Universal Robots PolyScope program: 8_put_glass_down.urp

Program 8_put_glass_down (installation=default directory=/programs/washer_rahman createdIn=5.9.5.1031259 lastSavedIn=5.9.5.1031259 robotSerialNumber=20215500597)
Calibrated DH parameters: a=[0.000193, -0.066673, -0.391568, -0.000012, 0.00005, 0]; d=[0.162643, -472.05677, 465.132521, 7.058239, 0.099746, 0.099582]; alpha=[1.571116, 0.00089, 0.003862, 1.569269, -1.569248, 0]; deltaTheta=[0, -1.413394, 7.628392, 0.068187, 0, -0.000001]
Robot Program (runOnlyOnce=true)
  SuppressedNode
    var_2 := 3
  SuppressedNode
    Script: glass_hover=p[-.603,-0.23+var_2*0.150 ,0.277,2.067,2.652,-2.043]
  Script: glass_hover=p[-.603,-0.23+GP_int_in[0]*0.150 ,0.277,2.067,2.652,-2.043]
  MoveJ speed 60 deg/s, acceleration 80 deg/s^2 (useActiveTCP=true) feature=Base
    Waypoint Waypoint_3: TCP in base x=-651.87 y=-69.028 z=453.929 mm, rx=-1.3447 ry=-1.3257 rz=0.979 rad; joints [-5.789, -92.229, 118.135, -194.029, -90.029, -4.694] deg; TCP offset x=0 y=0 z=191.5 mm, rx=0 ry=0 rz=0 rad
    SuppressedNode
      Waypoint Waypoint_4: TCP in base x=-472.073 y=-43.256 z=326.493 mm, rx=-1.3451 ry=-1.1695 rz=0.9064 rad; joints [-6.935, -98.689, 153.035, -227.002, -96.953, -4.705] deg
    SuppressedNode
      Waypoint Waypoint_2: TCP in base x=-651.885 y=-68.975 z=553.831 mm, rx=-1.3448 ry=-1.3258 rz=0.9788 rad; joints [-5.788, -96.752, 106.856, -178.218, -89.98, -4.691] deg
  SuppressedNode
    MoveJ speed 60 deg/s, acceleration 80 deg/s^2 (useActiveTCP=true) feature=Base
      SuppressedNode
        Waypoint Waypoint_1: TCP in base x=-651.863 y=-68.969 z=503.938 mm, rx=-1.3447 ry=-1.3257 rz=0.9789 rad; joints [-5.792, -95.02, 112.843, -185.947, -90.004, -4.691] deg
  MoveJ speed 60 deg/s, acceleration 80 deg/s^2 (useActiveTCP=true) feature=Base
    Waypoint Waypoint (Variable): variable=glass_hover
  MoveL speed 250 mm/s, acceleration 1200 mm/s^2 (useActiveTCP=true) feature=Base
    MoveDirectionNode (selectedDirection=ZMinus)
      Until DISTANCE (allowActions=false deceleration=3 distanceNodeType=STOP) Distance=0.18; motionParameters(blendRadius=0)
  URCap Gripper (Robotiq_Grippers, Robotiq Inc.) dataModel(position=15.294117647058822, force=0.0, speed=0.0, positionInDouble=15.294117647058822, forceInDouble=0.0, speedInDouble=0.0, slaveIds=[9], blocking=true)
  MoveL speed 250 mm/s, acceleration 1200 mm/s^2 (useActiveTCP=true) feature=Base
    MoveDirectionNode (selectedDirection=ZPlus)
      Until DISTANCE (allowActions=false deceleration=3 distanceNodeType=STOP) Distance=0.15; motionParameters(blendRadius=0)
  URCap Gripper (Robotiq_Grippers, Robotiq Inc.) dataModel(position=0.0, force=0.0, speed=0.0, positionInDouble=0.0, forceInDouble=0.0, speedInDouble=0.0, slaveIds=[9], blocking=true)
  MoveJ speed 60 deg/s, acceleration 80 deg/s^2 (useActiveTCP=true) feature=Base
    Waypoint Waypoint_1: TCP in base x=-557.948 y=-0.617 z=246.473 mm, rx=-1.2337 ry=-1.2229 rz=1.2356 rad; joints [-31.234, -63.252, 147.704, -263.239, -57.852, 1.051] deg
